INTERFACE I_OnlineChange EXTENDS I_Generic

METHOD OnOnlineChange
VAR_INPUT
	bEntityDeleted: BOOL;
	bEntityCreated: BOOL;
END_VAR
END_METHOD

END_INTERFACE

(* stored: Version 1.1.0.1
   Itf I_OnlineChange: Id {6cc3b00d-eb89-4fe3-9d4e-ba398a678a26}
   Method OnOnlineChange: Id {41955f3a-b1de-42fb-be12-ad92209e49a9} *)
